// TIA Portal V17 export
// export: Created 2025-03-05T07:58:51.8164485Z, ExportSetting WithDefaults, DisplayName Totally Integrated Automation Portal, DisplayVersion V17 Update 8, DisplayName TIA Portal Openness, DisplayVersion V17 Update 8, DisplayName TIA Portal Version Control Interface, DisplayVersion V17, DisplayName SINAMICS Startdrive Advanced, DisplayVersion V17 SP2, DisplayName SINAMICS Startdrive G110M, G120, G120C, G120D, G120P, G115D, DisplayVersion V17 SP2, DisplayName SINAMICS Startdrive G130, G150, S120, S150, SINAMICS MV, S210, DisplayVersion V17 SP2, DisplayName STEP 7 Professional, DisplayVersion V17 Update 8, DisplayName SINUMERIK ONE STEP 7 Toolbox, DisplayVersion V17 Update 12, DisplayName SINUMERIK 840D sl STEP 7 Toolbox, DisplayVersion V17 Update 12, DisplayName STEP 7 Safety, DisplayVersion V17 Update 6, DisplayName WinCC Advanced, DisplayVersion V17 Update 8
DATA_BLOCK "LBP_CtrlEnergy"   // DB1000
TITLE = Ctrl-Energy
{ S7_Optimized_Access := 'FALSE'; DB_Accessible_From_OPC_UA := 'FALSE' }
AUTHOR : SINUMERIK
FAMILY : SINUMERIK_ONE
VERSION : 6.15
// Interface between user program and operating software, contains energy-saving profiles for Ctrl-Energy / La interfaz entre programa de usuario y software operativo, contiene perfiles de ahorro energético para Ctrl-Energy / Schnittstelle zwischen Anwenderprogramm und Betriebssoftware, enthält energiesparende Profile für Ctrl-Energy
// stored: AutoNumber false, DBAccessibleFromOPCUA false, DBAccessibleFromWebserver true, IsOnlyStoredInLoadMemory false, IsWriteProtectedInAS false
   VAR RETAIN
      Profile : Array[1..8] of Struct
         ESaveOn : Bool;   // Energiesparendes Profil sofort aktivieren / Activate energy-saving profile immediately / Activar inmediatamente perfil de ahorro energético
         ReloadT2 : Bool;   // Vorwarnzeit (T2) neu laden / Reload Prewarning time (T2) / Volver a cargar tiempo de prealarma (T2)
         res0_2 : Bool;
         res0_3 : Bool;
         res0_4 : Bool;
         res0_5 : Bool;
         res0_6 : Bool;
         res0_7 : Bool;
         HmiESaveOn : Bool;   // HMI->PLC: Energiesparendes Profil sofort aktivieren / HMI->PLC: Activate energy-saving profile immediately / HMI->PLC: activar inmediatamente perfil de ahorro energético
         res1_1 : Bool;
         res1_2 : Bool;
         res1_3 : Bool;
         res1_4 : Bool;
         res1_5 : Bool;
         res1_6 : Bool;
         res1_7 : Bool;
         MasterCompSig : Bool;   // Master-Rechner-Signal / Master computer signal / Señal de equipo maestro
         PlcUserSig : Bool;   // PLC-Anwendersignal / PLC user signal / Señal de usuario PLC
         res2_2 : Bool;
         res2_3 : Bool;
         res2_4 : Bool;
         res2_5 : Bool;
         res2_6 : Bool;
         res2_7 : Bool;
         res3 : Byte;
         ESaveIsOn : Bool;   // Energiesparender Zustand aktiv / Energy-saving state active / Estado de ahorro energético activo
         T1Expired : Bool;   // Aktivierungszeit T1 abgelaufen / Activation time T1 expired / Tiempo de activación T1 agotado
         res4_2 : Bool;
         res4_3 : Bool;
         res4_4 : Bool;
         res4_5 : Bool;
         res4_6 : Bool;
         res4_7 : Bool;
         res5 : Byte;
         ActValT1 : Int;   // T1 aktueller Wert / T1 current value / T1 valor actual
         ActValT2 : Int;   // T2 aktueller Wert / T2 current value / T2 valor actual
         ESaveValid : Bool;   // HMI->PLC: Energiesparendes Profil gültig / HMI->PLC: Energy-saving profile valid / HMI->PLC: perfil de ahorro energético válido
         ESaveOff : Bool;   // HMI->PLC: Energiesparendes Profil deaktivieren/sperren / HMI->PLC: Deactivate energy-saving profileblock energy-saving profile / HMI->PLC: activar/desactivar perfil de ahorro energético
         res10_2 : Bool;
         res10_3 : Bool;
         res10_4 : Bool;
         res10_5 : Bool;
         res10_6 : Bool;
         res10_7 : Bool;
         CondOpPanel : Bool;   // HMI->PLC: Bedienfeld / HMI->PLC: Operator panel / HMI->PLC: panel de mando
         CondDataTransfer : Bool;   // HMI->PLC: Datenübertragung / HMI->PLC: Data transfer / HMI->PLC: transferencia de datos
         CondWindowChange : Bool;   // HMI->PLC: Fensterwechsel / HMI->PLC: Window change / HMI->PLC: cambio de ventana
         res11_3 : Bool;
         res11_4 : Bool;
         res11_5 : Bool;
         res11_6 : Bool;
         res11_7 : Bool;
         CondMCP : Bool;   // HMI->PLC: Maschinen-Bedienfeld / HMI->PLC: Machine control panel / HMI->PLC: panel de mando de máquina
         res12_1 : Bool;
         res12_2 : Bool;
         res12_3 : Bool;
         res12_4 : Bool;
         res12_5 : Bool;
         res12_6 : Bool;
         res12_7 : Bool;
         CondNcChan1 : Bool;   // HMI->PLC: NC-Kanal 1 in Reset / HMI->PLC: NC channel 1 in reset / HMI->PLC: canal CN 1 en reset
         CondNcChan2 : Bool;   // HMI->PLC: NC-Kanal 2 in Reset / HMI->PLC: NC channel 2 in reset / HMI->PLC: canal CN 2 en reset
         CondNcChan3 : Bool;   // HMI->PLC: NC-Kanal 3 in Reset / HMI->PLC: NC channel 3 in reset / HMI->PLC: canal CN 3 en reset
         CondNcChan4 : Bool;   // HMI->PLC: NC-Kanal 4 in Reset / HMI->PLC: NC channel 4 in reset / HMI->PLC: canal CN 4 en reset
         CondNcChan5 : Bool;   // HMI->PLC: NC-Kanal 5 in Reset / HMI->PLC: NC channel 5 in reset / HMI->PLC: canal CN 5 en reset
         CondNcChan6 : Bool;   // HMI->PLC: NC-Kanal 6 in Reset / HMI->PLC: NC channel 6 in reset / HMI->PLC: canal CN 6 en reset
         CondNcChan7 : Bool;   // HMI->PLC: NC-Kanal 7 in Reset / HMI->PLC: NC channel 7 in reset / HMI->PLC: canal CN 7 en reset
         CondNcChan8 : Bool;   // HMI->PLC: NC-Kanal 8 in Reset / HMI->PLC: NC channel 8 in reset / HMI->PLC: canal CN 8 en reset
         CondNcChan9 : Bool;   // HMI->PLC: NC-Kanal 9 in Reset / HMI->PLC: NC channel 9 in reset / HMI->PLC: canal CN 9 en reset
         CondNcChan10 : Bool;   // HMI->PLC: NC-Kanal 10 in Reset / HMI->PLC: NC channel 10 in reset / HMI->PLC: canal CN 10 en reset
         res14_2 : Bool;
         res14_3 : Bool;
         res14_4 : Bool;
         res14_5 : Bool;
         res14_6 : Bool;
         res14_7 : Bool;
         CondMasterCompSig : Bool;   // HMI->PLC: Master-Rechner-Signal / HMI->PLC: Master computer signal / HMI->PLC: señal de equipo maestro
         CondPlcUserSig : Bool;   // HMI->PLC: PLC-Anwendersignal / HMI->PLC: PLC user signal / HMI->PLC: señal de usuario PLC
         res15_2 : Bool;
         res15_3 : Bool;
         res15_4 : Bool;
         res15_5 : Bool;
         res15_6 : Bool;
         res15_7 : Bool;
         PresetT1 : Int;   // HMI->PLC: Aktivierung Zeit T1 / HMI->PLC: Activation time T1 / HMI->PLC: activación tiempo T1
         PresetT2 : Int;   // HMI->PLC: Vorwarnzeit T2 / HMI->PLC: Prewarning time T2 / HMI->PLC: tiempo de prealarma T2
      END_STRUCT;
   END_VAR
BEGIN
   // Profile[2].ESaveOn : Energiesparendes Profil sofort aktivieren / Activate energy-saving profile immediately / Activar inmediatamente perfil de ahorro energético
   // Profile[3].ESaveOn : Energiesparendes Profil sofort aktivieren / Activate energy-saving profile immediately / Activar inmediatamente perfil de ahorro energético
   // Profile[4].ESaveOn : Energiesparendes Profil sofort aktivieren / Activate energy-saving profile immediately / Activar inmediatamente perfil de ahorro energético
   // Profile[5].ESaveOn : Energiesparendes Profil sofort aktivieren / Activate energy-saving profile immediately / Activar inmediatamente perfil de ahorro energético
   // Profile[6].ESaveOn : Energiesparendes Profil sofort aktivieren / Activate energy-saving profile immediately / Activar inmediatamente perfil de ahorro energético
   // Profile[7].ESaveOn : Energiesparendes Profil sofort aktivieren / Activate energy-saving profile immediately / Activar inmediatamente perfil de ahorro energético
   // Profile[8].ESaveOn : Energiesparendes Profil sofort aktivieren / Activate energy-saving profile immediately / Activar inmediatamente perfil de ahorro energético
   // Profile[2].ReloadT2 : Vorwarnzeit (T2) neu laden / Reload Prewarning time (T2) / Volver a cargar tiempo de prealarma (T2)
   // Profile[3].ReloadT2 : Vorwarnzeit (T2) neu laden / Reload Prewarning time (T2) / Volver a cargar tiempo de prealarma (T2)
   // Profile[4].ReloadT2 : Vorwarnzeit (T2) neu laden / Reload Prewarning time (T2) / Volver a cargar tiempo de prealarma (T2)
   // Profile[5].ReloadT2 : Vorwarnzeit (T2) neu laden / Reload Prewarning time (T2) / Volver a cargar tiempo de prealarma (T2)
   // Profile[6].ReloadT2 : Vorwarnzeit (T2) neu laden / Reload Prewarning time (T2) / Volver a cargar tiempo de prealarma (T2)
   // Profile[7].ReloadT2 : Vorwarnzeit (T2) neu laden / Reload Prewarning time (T2) / Volver a cargar tiempo de prealarma (T2)
   // Profile[8].ReloadT2 : Vorwarnzeit (T2) neu laden / Reload Prewarning time (T2) / Volver a cargar tiempo de prealarma (T2)
   // Profile[2].HmiESaveOn : HMI->PLC: Energiesparendes Profil sofort aktivieren / HMI->PLC: Activate energy-saving profile immediately / HMI->PLC: activar inmediatamente perfil de ahorro energético
   // Profile[3].HmiESaveOn : HMI->PLC: Energiesparendes Profil sofort aktivieren / HMI->PLC: Activate energy-saving profile immediately / HMI->PLC: activar inmediatamente perfil de ahorro energético
   // Profile[4].HmiESaveOn : HMI->PLC: Energiesparendes Profil sofort aktivieren / HMI->PLC: Activate energy-saving profile immediately / HMI->PLC: activar inmediatamente perfil de ahorro energético
   // Profile[5].HmiESaveOn : HMI->PLC: Energiesparendes Profil sofort aktivieren / HMI->PLC: Activate energy-saving profile immediately / HMI->PLC: activar inmediatamente perfil de ahorro energético
   // Profile[6].HmiESaveOn : HMI->PLC: Energiesparendes Profil sofort aktivieren / HMI->PLC: Activate energy-saving profile immediately / HMI->PLC: activar inmediatamente perfil de ahorro energético
   // Profile[7].HmiESaveOn : HMI->PLC: Energiesparendes Profil sofort aktivieren / HMI->PLC: Activate energy-saving profile immediately / HMI->PLC: activar inmediatamente perfil de ahorro energético
   // Profile[8].HmiESaveOn : HMI->PLC: Energiesparendes Profil sofort aktivieren / HMI->PLC: Activate energy-saving profile immediately / HMI->PLC: activar inmediatamente perfil de ahorro energético
   // Profile[2].MasterCompSig : Master-Rechner-Signal / Master computer signal / Señal de equipo maestro
   // Profile[3].MasterCompSig : Master-Rechner-Signal / Master computer signal / Señal de equipo maestro
   // Profile[4].MasterCompSig : Master-Rechner-Signal / Master computer signal / Señal de equipo maestro
   // Profile[5].MasterCompSig : Master-Rechner-Signal / Master computer signal / Señal de equipo maestro
   // Profile[6].MasterCompSig : Master-Rechner-Signal / Master computer signal / Señal de equipo maestro
   // Profile[7].MasterCompSig : Master-Rechner-Signal / Master computer signal / Señal de equipo maestro
   // Profile[8].MasterCompSig : Master-Rechner-Signal / Master computer signal / Señal de equipo maestro
   // Profile[2].PlcUserSig : PLC-Anwendersignal / PLC user signal / Señal de usuario PLC
   // Profile[3].PlcUserSig : PLC-Anwendersignal / PLC user signal / Señal de usuario PLC
   // Profile[4].PlcUserSig : PLC-Anwendersignal / PLC user signal / Señal de usuario PLC
   // Profile[5].PlcUserSig : PLC-Anwendersignal / PLC user signal / Señal de usuario PLC
   // Profile[6].PlcUserSig : PLC-Anwendersignal / PLC user signal / Señal de usuario PLC
   // Profile[7].PlcUserSig : PLC-Anwendersignal / PLC user signal / Señal de usuario PLC
   // Profile[8].PlcUserSig : PLC-Anwendersignal / PLC user signal / Señal de usuario PLC
   // Profile[2].ESaveIsOn : Energiesparender Zustand aktiv / Energy-saving state active / Estado de ahorro energético activo
   // Profile[3].ESaveIsOn : Energiesparender Zustand aktiv / Energy-saving state active / Estado de ahorro energético activo
   // Profile[4].ESaveIsOn : Energiesparender Zustand aktiv / Energy-saving state active / Estado de ahorro energético activo
   // Profile[5].ESaveIsOn : Energiesparender Zustand aktiv / Energy-saving state active / Estado de ahorro energético activo
   // Profile[6].ESaveIsOn : Energiesparender Zustand aktiv / Energy-saving state active / Estado de ahorro energético activo
   // Profile[7].ESaveIsOn : Energiesparender Zustand aktiv / Energy-saving state active / Estado de ahorro energético activo
   // Profile[8].ESaveIsOn : Energiesparender Zustand aktiv / Energy-saving state active / Estado de ahorro energético activo
   // Profile[2].T1Expired : Aktivierungszeit T1 abgelaufen / Activation time T1 expired / Tiempo de activación T1 agotado
   // Profile[3].T1Expired : Aktivierungszeit T1 abgelaufen / Activation time T1 expired / Tiempo de activación T1 agotado
   // Profile[4].T1Expired : Aktivierungszeit T1 abgelaufen / Activation time T1 expired / Tiempo de activación T1 agotado
   // Profile[5].T1Expired : Aktivierungszeit T1 abgelaufen / Activation time T1 expired / Tiempo de activación T1 agotado
   // Profile[6].T1Expired : Aktivierungszeit T1 abgelaufen / Activation time T1 expired / Tiempo de activación T1 agotado
   // Profile[7].T1Expired : Aktivierungszeit T1 abgelaufen / Activation time T1 expired / Tiempo de activación T1 agotado
   // Profile[8].T1Expired : Aktivierungszeit T1 abgelaufen / Activation time T1 expired / Tiempo de activación T1 agotado
   // Profile[2].ActValT1 : T1 aktueller Wert / T1 current value / T1 valor actual
   // Profile[3].ActValT1 : T1 aktueller Wert / T1 current value / T1 valor actual
   // Profile[4].ActValT1 : T1 aktueller Wert / T1 current value / T1 valor actual
   // Profile[5].ActValT1 : T1 aktueller Wert / T1 current value / T1 valor actual
   // Profile[6].ActValT1 : T1 aktueller Wert / T1 current value / T1 valor actual
   // Profile[7].ActValT1 : T1 aktueller Wert / T1 current value / T1 valor actual
   // Profile[8].ActValT1 : T1 aktueller Wert / T1 current value / T1 valor actual
   // Profile[2].ActValT2 : T2 aktueller Wert / T2 current value / T2 valor actual
   // Profile[3].ActValT2 : T2 aktueller Wert / T2 current value / T2 valor actual
   // Profile[4].ActValT2 : T2 aktueller Wert / T2 current value / T2 valor actual
   // Profile[5].ActValT2 : T2 aktueller Wert / T2 current value / T2 valor actual
   // Profile[6].ActValT2 : T2 aktueller Wert / T2 current value / T2 valor actual
   // Profile[7].ActValT2 : T2 aktueller Wert / T2 current value / T2 valor actual
   // Profile[8].ActValT2 : T2 aktueller Wert / T2 current value / T2 valor actual
   Profile[1].ESaveValid := TRUE;
   Profile[2].ESaveValid := TRUE;   // HMI->PLC: Energiesparendes Profil gültig / HMI->PLC: Energy-saving profile valid / HMI->PLC: perfil de ahorro energético válido
   Profile[3].ESaveValid := TRUE;   // HMI->PLC: Energiesparendes Profil gültig / HMI->PLC: Energy-saving profile valid / HMI->PLC: perfil de ahorro energético válido
   // Profile[4].ESaveValid : HMI->PLC: Energiesparendes Profil gültig / HMI->PLC: Energy-saving profile valid / HMI->PLC: perfil de ahorro energético válido
   // Profile[5].ESaveValid : HMI->PLC: Energiesparendes Profil gültig / HMI->PLC: Energy-saving profile valid / HMI->PLC: perfil de ahorro energético válido
   // Profile[6].ESaveValid : HMI->PLC: Energiesparendes Profil gültig / HMI->PLC: Energy-saving profile valid / HMI->PLC: perfil de ahorro energético válido
   // Profile[7].ESaveValid : HMI->PLC: Energiesparendes Profil gültig / HMI->PLC: Energy-saving profile valid / HMI->PLC: perfil de ahorro energético válido
   // Profile[8].ESaveValid : HMI->PLC: Energiesparendes Profil gültig / HMI->PLC: Energy-saving profile valid / HMI->PLC: perfil de ahorro energético válido
   Profile[1].ESaveOff := TRUE;
   Profile[2].ESaveOff := TRUE;   // HMI->PLC: Energiesparendes Profil deaktivieren/sperren / HMI->PLC: Deactivate energy-saving profileblock energy-saving profile / HMI->PLC: activar/desactivar perfil de ahorro energético
   Profile[3].ESaveOff := TRUE;   // HMI->PLC: Energiesparendes Profil deaktivieren/sperren / HMI->PLC: Deactivate energy-saving profileblock energy-saving profile / HMI->PLC: activar/desactivar perfil de ahorro energético
   // Profile[4].ESaveOff : HMI->PLC: Energiesparendes Profil deaktivieren/sperren / HMI->PLC: Deactivate energy-saving profileblock energy-saving profile / HMI->PLC: activar/desactivar perfil de ahorro energético
   // Profile[5].ESaveOff : HMI->PLC: Energiesparendes Profil deaktivieren/sperren / HMI->PLC: Deactivate energy-saving profileblock energy-saving profile / HMI->PLC: activar/desactivar perfil de ahorro energético
   // Profile[6].ESaveOff : HMI->PLC: Energiesparendes Profil deaktivieren/sperren / HMI->PLC: Deactivate energy-saving profileblock energy-saving profile / HMI->PLC: activar/desactivar perfil de ahorro energético
   // Profile[7].ESaveOff : HMI->PLC: Energiesparendes Profil deaktivieren/sperren / HMI->PLC: Deactivate energy-saving profileblock energy-saving profile / HMI->PLC: activar/desactivar perfil de ahorro energético
   // Profile[8].ESaveOff : HMI->PLC: Energiesparendes Profil deaktivieren/sperren / HMI->PLC: Deactivate energy-saving profileblock energy-saving profile / HMI->PLC: activar/desactivar perfil de ahorro energético
   // Profile[2].CondOpPanel : HMI->PLC: Bedienfeld / HMI->PLC: Operator panel / HMI->PLC: panel de mando
   Profile[3].CondOpPanel := TRUE;   // HMI->PLC: Bedienfeld / HMI->PLC: Operator panel / HMI->PLC: panel de mando
   // Profile[4].CondOpPanel : HMI->PLC: Bedienfeld / HMI->PLC: Operator panel / HMI->PLC: panel de mando
   // Profile[5].CondOpPanel : HMI->PLC: Bedienfeld / HMI->PLC: Operator panel / HMI->PLC: panel de mando
   // Profile[6].CondOpPanel : HMI->PLC: Bedienfeld / HMI->PLC: Operator panel / HMI->PLC: panel de mando
   // Profile[7].CondOpPanel : HMI->PLC: Bedienfeld / HMI->PLC: Operator panel / HMI->PLC: panel de mando
   // Profile[8].CondOpPanel : HMI->PLC: Bedienfeld / HMI->PLC: Operator panel / HMI->PLC: panel de mando
   // Profile[2].CondDataTransfer : HMI->PLC: Datenübertragung / HMI->PLC: Data transfer / HMI->PLC: transferencia de datos
   Profile[3].CondDataTransfer := TRUE;   // HMI->PLC: Datenübertragung / HMI->PLC: Data transfer / HMI->PLC: transferencia de datos
   // Profile[4].CondDataTransfer : HMI->PLC: Datenübertragung / HMI->PLC: Data transfer / HMI->PLC: transferencia de datos
   // Profile[5].CondDataTransfer : HMI->PLC: Datenübertragung / HMI->PLC: Data transfer / HMI->PLC: transferencia de datos
   // Profile[6].CondDataTransfer : HMI->PLC: Datenübertragung / HMI->PLC: Data transfer / HMI->PLC: transferencia de datos
   // Profile[7].CondDataTransfer : HMI->PLC: Datenübertragung / HMI->PLC: Data transfer / HMI->PLC: transferencia de datos
   // Profile[8].CondDataTransfer : HMI->PLC: Datenübertragung / HMI->PLC: Data transfer / HMI->PLC: transferencia de datos
   // Profile[2].CondWindowChange : HMI->PLC: Fensterwechsel / HMI->PLC: Window change / HMI->PLC: cambio de ventana
   Profile[3].CondWindowChange := TRUE;   // HMI->PLC: Fensterwechsel / HMI->PLC: Window change / HMI->PLC: cambio de ventana
   // Profile[4].CondWindowChange : HMI->PLC: Fensterwechsel / HMI->PLC: Window change / HMI->PLC: cambio de ventana
   // Profile[5].CondWindowChange : HMI->PLC: Fensterwechsel / HMI->PLC: Window change / HMI->PLC: cambio de ventana
   // Profile[6].CondWindowChange : HMI->PLC: Fensterwechsel / HMI->PLC: Window change / HMI->PLC: cambio de ventana
   // Profile[7].CondWindowChange : HMI->PLC: Fensterwechsel / HMI->PLC: Window change / HMI->PLC: cambio de ventana
   // Profile[8].CondWindowChange : HMI->PLC: Fensterwechsel / HMI->PLC: Window change / HMI->PLC: cambio de ventana
   Profile[2].CondMCP := TRUE;   // HMI->PLC: Maschinen-Bedienfeld / HMI->PLC: Machine control panel / HMI->PLC: panel de mando de máquina
   Profile[3].CondMCP := TRUE;   // HMI->PLC: Maschinen-Bedienfeld / HMI->PLC: Machine control panel / HMI->PLC: panel de mando de máquina
   // Profile[4].CondMCP : HMI->PLC: Maschinen-Bedienfeld / HMI->PLC: Machine control panel / HMI->PLC: panel de mando de máquina
   // Profile[5].CondMCP : HMI->PLC: Maschinen-Bedienfeld / HMI->PLC: Machine control panel / HMI->PLC: panel de mando de máquina
   // Profile[6].CondMCP : HMI->PLC: Maschinen-Bedienfeld / HMI->PLC: Machine control panel / HMI->PLC: panel de mando de máquina
   // Profile[7].CondMCP : HMI->PLC: Maschinen-Bedienfeld / HMI->PLC: Machine control panel / HMI->PLC: panel de mando de máquina
   // Profile[8].CondMCP : HMI->PLC: Maschinen-Bedienfeld / HMI->PLC: Machine control panel / HMI->PLC: panel de mando de máquina
   Profile[1].CondNcChan1 := TRUE;
   Profile[2].CondNcChan1 := TRUE;   // HMI->PLC: NC-Kanal 1 in Reset / HMI->PLC: NC channel 1 in reset / HMI->PLC: canal CN 1 en reset
   Profile[3].CondNcChan1 := TRUE;   // HMI->PLC: NC-Kanal 1 in Reset / HMI->PLC: NC channel 1 in reset / HMI->PLC: canal CN 1 en reset
   // Profile[4].CondNcChan1 : HMI->PLC: NC-Kanal 1 in Reset / HMI->PLC: NC channel 1 in reset / HMI->PLC: canal CN 1 en reset
   // Profile[5].CondNcChan1 : HMI->PLC: NC-Kanal 1 in Reset / HMI->PLC: NC channel 1 in reset / HMI->PLC: canal CN 1 en reset
   // Profile[6].CondNcChan1 : HMI->PLC: NC-Kanal 1 in Reset / HMI->PLC: NC channel 1 in reset / HMI->PLC: canal CN 1 en reset
   // Profile[7].CondNcChan1 : HMI->PLC: NC-Kanal 1 in Reset / HMI->PLC: NC channel 1 in reset / HMI->PLC: canal CN 1 en reset
   // Profile[8].CondNcChan1 : HMI->PLC: NC-Kanal 1 in Reset / HMI->PLC: NC channel 1 in reset / HMI->PLC: canal CN 1 en reset
   Profile[1].CondNcChan2 := TRUE;
   Profile[2].CondNcChan2 := TRUE;   // HMI->PLC: NC-Kanal 2 in Reset / HMI->PLC: NC channel 2 in reset / HMI->PLC: canal CN 2 en reset
   Profile[3].CondNcChan2 := TRUE;   // HMI->PLC: NC-Kanal 2 in Reset / HMI->PLC: NC channel 2 in reset / HMI->PLC: canal CN 2 en reset
   // Profile[4].CondNcChan2 : HMI->PLC: NC-Kanal 2 in Reset / HMI->PLC: NC channel 2 in reset / HMI->PLC: canal CN 2 en reset
   // Profile[5].CondNcChan2 : HMI->PLC: NC-Kanal 2 in Reset / HMI->PLC: NC channel 2 in reset / HMI->PLC: canal CN 2 en reset
   // Profile[6].CondNcChan2 : HMI->PLC: NC-Kanal 2 in Reset / HMI->PLC: NC channel 2 in reset / HMI->PLC: canal CN 2 en reset
   // Profile[7].CondNcChan2 : HMI->PLC: NC-Kanal 2 in Reset / HMI->PLC: NC channel 2 in reset / HMI->PLC: canal CN 2 en reset
   // Profile[8].CondNcChan2 : HMI->PLC: NC-Kanal 2 in Reset / HMI->PLC: NC channel 2 in reset / HMI->PLC: canal CN 2 en reset
   Profile[1].CondNcChan3 := TRUE;
   Profile[2].CondNcChan3 := TRUE;   // HMI->PLC: NC-Kanal 3 in Reset / HMI->PLC: NC channel 3 in reset / HMI->PLC: canal CN 3 en reset
   Profile[3].CondNcChan3 := TRUE;   // HMI->PLC: NC-Kanal 3 in Reset / HMI->PLC: NC channel 3 in reset / HMI->PLC: canal CN 3 en reset
   // Profile[4].CondNcChan3 : HMI->PLC: NC-Kanal 3 in Reset / HMI->PLC: NC channel 3 in reset / HMI->PLC: canal CN 3 en reset
   // Profile[5].CondNcChan3 : HMI->PLC: NC-Kanal 3 in Reset / HMI->PLC: NC channel 3 in reset / HMI->PLC: canal CN 3 en reset
   // Profile[6].CondNcChan3 : HMI->PLC: NC-Kanal 3 in Reset / HMI->PLC: NC channel 3 in reset / HMI->PLC: canal CN 3 en reset
   // Profile[7].CondNcChan3 : HMI->PLC: NC-Kanal 3 in Reset / HMI->PLC: NC channel 3 in reset / HMI->PLC: canal CN 3 en reset
   // Profile[8].CondNcChan3 : HMI->PLC: NC-Kanal 3 in Reset / HMI->PLC: NC channel 3 in reset / HMI->PLC: canal CN 3 en reset
   Profile[1].CondNcChan4 := TRUE;
   Profile[2].CondNcChan4 := TRUE;   // HMI->PLC: NC-Kanal 4 in Reset / HMI->PLC: NC channel 4 in reset / HMI->PLC: canal CN 4 en reset
   Profile[3].CondNcChan4 := TRUE;   // HMI->PLC: NC-Kanal 4 in Reset / HMI->PLC: NC channel 4 in reset / HMI->PLC: canal CN 4 en reset
   // Profile[4].CondNcChan4 : HMI->PLC: NC-Kanal 4 in Reset / HMI->PLC: NC channel 4 in reset / HMI->PLC: canal CN 4 en reset
   // Profile[5].CondNcChan4 : HMI->PLC: NC-Kanal 4 in Reset / HMI->PLC: NC channel 4 in reset / HMI->PLC: canal CN 4 en reset
   // Profile[6].CondNcChan4 : HMI->PLC: NC-Kanal 4 in Reset / HMI->PLC: NC channel 4 in reset / HMI->PLC: canal CN 4 en reset
   // Profile[7].CondNcChan4 : HMI->PLC: NC-Kanal 4 in Reset / HMI->PLC: NC channel 4 in reset / HMI->PLC: canal CN 4 en reset
   // Profile[8].CondNcChan4 : HMI->PLC: NC-Kanal 4 in Reset / HMI->PLC: NC channel 4 in reset / HMI->PLC: canal CN 4 en reset
   Profile[1].CondNcChan5 := TRUE;
   Profile[2].CondNcChan5 := TRUE;   // HMI->PLC: NC-Kanal 5 in Reset / HMI->PLC: NC channel 5 in reset / HMI->PLC: canal CN 5 en reset
   Profile[3].CondNcChan5 := TRUE;   // HMI->PLC: NC-Kanal 5 in Reset / HMI->PLC: NC channel 5 in reset / HMI->PLC: canal CN 5 en reset
   // Profile[4].CondNcChan5 : HMI->PLC: NC-Kanal 5 in Reset / HMI->PLC: NC channel 5 in reset / HMI->PLC: canal CN 5 en reset
   // Profile[5].CondNcChan5 : HMI->PLC: NC-Kanal 5 in Reset / HMI->PLC: NC channel 5 in reset / HMI->PLC: canal CN 5 en reset
   // Profile[6].CondNcChan5 : HMI->PLC: NC-Kanal 5 in Reset / HMI->PLC: NC channel 5 in reset / HMI->PLC: canal CN 5 en reset
   // Profile[7].CondNcChan5 : HMI->PLC: NC-Kanal 5 in Reset / HMI->PLC: NC channel 5 in reset / HMI->PLC: canal CN 5 en reset
   // Profile[8].CondNcChan5 : HMI->PLC: NC-Kanal 5 in Reset / HMI->PLC: NC channel 5 in reset / HMI->PLC: canal CN 5 en reset
   Profile[1].CondNcChan6 := TRUE;
   Profile[2].CondNcChan6 := TRUE;   // HMI->PLC: NC-Kanal 6 in Reset / HMI->PLC: NC channel 6 in reset / HMI->PLC: canal CN 6 en reset
   Profile[3].CondNcChan6 := TRUE;   // HMI->PLC: NC-Kanal 6 in Reset / HMI->PLC: NC channel 6 in reset / HMI->PLC: canal CN 6 en reset
   // Profile[4].CondNcChan6 : HMI->PLC: NC-Kanal 6 in Reset / HMI->PLC: NC channel 6 in reset / HMI->PLC: canal CN 6 en reset
   // Profile[5].CondNcChan6 : HMI->PLC: NC-Kanal 6 in Reset / HMI->PLC: NC channel 6 in reset / HMI->PLC: canal CN 6 en reset
   // Profile[6].CondNcChan6 : HMI->PLC: NC-Kanal 6 in Reset / HMI->PLC: NC channel 6 in reset / HMI->PLC: canal CN 6 en reset
   // Profile[7].CondNcChan6 : HMI->PLC: NC-Kanal 6 in Reset / HMI->PLC: NC channel 6 in reset / HMI->PLC: canal CN 6 en reset
   // Profile[8].CondNcChan6 : HMI->PLC: NC-Kanal 6 in Reset / HMI->PLC: NC channel 6 in reset / HMI->PLC: canal CN 6 en reset
   Profile[1].CondNcChan7 := TRUE;
   Profile[2].CondNcChan7 := TRUE;   // HMI->PLC: NC-Kanal 7 in Reset / HMI->PLC: NC channel 7 in reset / HMI->PLC: canal CN 7 en reset
   Profile[3].CondNcChan7 := TRUE;   // HMI->PLC: NC-Kanal 7 in Reset / HMI->PLC: NC channel 7 in reset / HMI->PLC: canal CN 7 en reset
   // Profile[4].CondNcChan7 : HMI->PLC: NC-Kanal 7 in Reset / HMI->PLC: NC channel 7 in reset / HMI->PLC: canal CN 7 en reset
   // Profile[5].CondNcChan7 : HMI->PLC: NC-Kanal 7 in Reset / HMI->PLC: NC channel 7 in reset / HMI->PLC: canal CN 7 en reset
   // Profile[6].CondNcChan7 : HMI->PLC: NC-Kanal 7 in Reset / HMI->PLC: NC channel 7 in reset / HMI->PLC: canal CN 7 en reset
   // Profile[7].CondNcChan7 : HMI->PLC: NC-Kanal 7 in Reset / HMI->PLC: NC channel 7 in reset / HMI->PLC: canal CN 7 en reset
   // Profile[8].CondNcChan7 : HMI->PLC: NC-Kanal 7 in Reset / HMI->PLC: NC channel 7 in reset / HMI->PLC: canal CN 7 en reset
   Profile[1].CondNcChan8 := TRUE;
   Profile[2].CondNcChan8 := TRUE;   // HMI->PLC: NC-Kanal 8 in Reset / HMI->PLC: NC channel 8 in reset / HMI->PLC: canal CN 8 en reset
   Profile[3].CondNcChan8 := TRUE;   // HMI->PLC: NC-Kanal 8 in Reset / HMI->PLC: NC channel 8 in reset / HMI->PLC: canal CN 8 en reset
   // Profile[4].CondNcChan8 : HMI->PLC: NC-Kanal 8 in Reset / HMI->PLC: NC channel 8 in reset / HMI->PLC: canal CN 8 en reset
   // Profile[5].CondNcChan8 : HMI->PLC: NC-Kanal 8 in Reset / HMI->PLC: NC channel 8 in reset / HMI->PLC: canal CN 8 en reset
   // Profile[6].CondNcChan8 : HMI->PLC: NC-Kanal 8 in Reset / HMI->PLC: NC channel 8 in reset / HMI->PLC: canal CN 8 en reset
   // Profile[7].CondNcChan8 : HMI->PLC: NC-Kanal 8 in Reset / HMI->PLC: NC channel 8 in reset / HMI->PLC: canal CN 8 en reset
   // Profile[8].CondNcChan8 : HMI->PLC: NC-Kanal 8 in Reset / HMI->PLC: NC channel 8 in reset / HMI->PLC: canal CN 8 en reset
   Profile[1].CondNcChan9 := TRUE;
   Profile[2].CondNcChan9 := TRUE;   // HMI->PLC: NC-Kanal 9 in Reset / HMI->PLC: NC channel 9 in reset / HMI->PLC: canal CN 9 en reset
   Profile[3].CondNcChan9 := TRUE;   // HMI->PLC: NC-Kanal 9 in Reset / HMI->PLC: NC channel 9 in reset / HMI->PLC: canal CN 9 en reset
   // Profile[4].CondNcChan9 : HMI->PLC: NC-Kanal 9 in Reset / HMI->PLC: NC channel 9 in reset / HMI->PLC: canal CN 9 en reset
   // Profile[5].CondNcChan9 : HMI->PLC: NC-Kanal 9 in Reset / HMI->PLC: NC channel 9 in reset / HMI->PLC: canal CN 9 en reset
   // Profile[6].CondNcChan9 : HMI->PLC: NC-Kanal 9 in Reset / HMI->PLC: NC channel 9 in reset / HMI->PLC: canal CN 9 en reset
   // Profile[7].CondNcChan9 : HMI->PLC: NC-Kanal 9 in Reset / HMI->PLC: NC channel 9 in reset / HMI->PLC: canal CN 9 en reset
   // Profile[8].CondNcChan9 : HMI->PLC: NC-Kanal 9 in Reset / HMI->PLC: NC channel 9 in reset / HMI->PLC: canal CN 9 en reset
   Profile[1].CondNcChan10 := TRUE;
   Profile[2].CondNcChan10 := TRUE;   // HMI->PLC: NC-Kanal 10 in Reset / HMI->PLC: NC channel 10 in reset / HMI->PLC: canal CN 10 en reset
   Profile[3].CondNcChan10 := TRUE;   // HMI->PLC: NC-Kanal 10 in Reset / HMI->PLC: NC channel 10 in reset / HMI->PLC: canal CN 10 en reset
   // Profile[4].CondNcChan10 : HMI->PLC: NC-Kanal 10 in Reset / HMI->PLC: NC channel 10 in reset / HMI->PLC: canal CN 10 en reset
   // Profile[5].CondNcChan10 : HMI->PLC: NC-Kanal 10 in Reset / HMI->PLC: NC channel 10 in reset / HMI->PLC: canal CN 10 en reset
   // Profile[6].CondNcChan10 : HMI->PLC: NC-Kanal 10 in Reset / HMI->PLC: NC channel 10 in reset / HMI->PLC: canal CN 10 en reset
   // Profile[7].CondNcChan10 : HMI->PLC: NC-Kanal 10 in Reset / HMI->PLC: NC channel 10 in reset / HMI->PLC: canal CN 10 en reset
   // Profile[8].CondNcChan10 : HMI->PLC: NC-Kanal 10 in Reset / HMI->PLC: NC channel 10 in reset / HMI->PLC: canal CN 10 en reset
   // Profile[2].CondMasterCompSig : HMI->PLC: Master-Rechner-Signal / HMI->PLC: Master computer signal / HMI->PLC: señal de equipo maestro
   // Profile[3].CondMasterCompSig : HMI->PLC: Master-Rechner-Signal / HMI->PLC: Master computer signal / HMI->PLC: señal de equipo maestro
   // Profile[4].CondMasterCompSig : HMI->PLC: Master-Rechner-Signal / HMI->PLC: Master computer signal / HMI->PLC: señal de equipo maestro
   // Profile[5].CondMasterCompSig : HMI->PLC: Master-Rechner-Signal / HMI->PLC: Master computer signal / HMI->PLC: señal de equipo maestro
   // Profile[6].CondMasterCompSig : HMI->PLC: Master-Rechner-Signal / HMI->PLC: Master computer signal / HMI->PLC: señal de equipo maestro
   // Profile[7].CondMasterCompSig : HMI->PLC: Master-Rechner-Signal / HMI->PLC: Master computer signal / HMI->PLC: señal de equipo maestro
   // Profile[8].CondMasterCompSig : HMI->PLC: Master-Rechner-Signal / HMI->PLC: Master computer signal / HMI->PLC: señal de equipo maestro
   Profile[1].CondPlcUserSig := TRUE;
   Profile[2].CondPlcUserSig := TRUE;   // HMI->PLC: PLC-Anwendersignal / HMI->PLC: PLC user signal / HMI->PLC: señal de usuario PLC
   Profile[3].CondPlcUserSig := TRUE;   // HMI->PLC: PLC-Anwendersignal / HMI->PLC: PLC user signal / HMI->PLC: señal de usuario PLC
   // Profile[4].CondPlcUserSig : HMI->PLC: PLC-Anwendersignal / HMI->PLC: PLC user signal / HMI->PLC: señal de usuario PLC
   // Profile[5].CondPlcUserSig : HMI->PLC: PLC-Anwendersignal / HMI->PLC: PLC user signal / HMI->PLC: señal de usuario PLC
   // Profile[6].CondPlcUserSig : HMI->PLC: PLC-Anwendersignal / HMI->PLC: PLC user signal / HMI->PLC: señal de usuario PLC
   // Profile[7].CondPlcUserSig : HMI->PLC: PLC-Anwendersignal / HMI->PLC: PLC user signal / HMI->PLC: señal de usuario PLC
   // Profile[8].CondPlcUserSig : HMI->PLC: PLC-Anwendersignal / HMI->PLC: PLC user signal / HMI->PLC: señal de usuario PLC
   Profile[1].PresetT1 := 60;
   Profile[2].PresetT1 := 120;   // HMI->PLC: Aktivierung Zeit T1 / HMI->PLC: Activation time T1 / HMI->PLC: activación tiempo T1
   Profile[3].PresetT1 := 600;   // HMI->PLC: Aktivierung Zeit T1 / HMI->PLC: Activation time T1 / HMI->PLC: activación tiempo T1
   // Profile[4].PresetT1 : HMI->PLC: Aktivierung Zeit T1 / HMI->PLC: Activation time T1 / HMI->PLC: activación tiempo T1
   // Profile[5].PresetT1 : HMI->PLC: Aktivierung Zeit T1 / HMI->PLC: Activation time T1 / HMI->PLC: activación tiempo T1
   // Profile[6].PresetT1 : HMI->PLC: Aktivierung Zeit T1 / HMI->PLC: Activation time T1 / HMI->PLC: activación tiempo T1
   // Profile[7].PresetT1 : HMI->PLC: Aktivierung Zeit T1 / HMI->PLC: Activation time T1 / HMI->PLC: activación tiempo T1
   // Profile[8].PresetT1 : HMI->PLC: Aktivierung Zeit T1 / HMI->PLC: Activation time T1 / HMI->PLC: activación tiempo T1
   Profile[1].PresetT2 := 120;
   Profile[2].PresetT2 := 300;   // HMI->PLC: Vorwarnzeit T2 / HMI->PLC: Prewarning time T2 / HMI->PLC: tiempo de prealarma T2
   // Profile[3].PresetT2 : HMI->PLC: Vorwarnzeit T2 / HMI->PLC: Prewarning time T2 / HMI->PLC: tiempo de prealarma T2
   // Profile[4].PresetT2 : HMI->PLC: Vorwarnzeit T2 / HMI->PLC: Prewarning time T2 / HMI->PLC: tiempo de prealarma T2
   // Profile[5].PresetT2 : HMI->PLC: Vorwarnzeit T2 / HMI->PLC: Prewarning time T2 / HMI->PLC: tiempo de prealarma T2
   // Profile[6].PresetT2 : HMI->PLC: Vorwarnzeit T2 / HMI->PLC: Prewarning time T2 / HMI->PLC: tiempo de prealarma T2
   // Profile[7].PresetT2 : HMI->PLC: Vorwarnzeit T2 / HMI->PLC: Prewarning time T2 / HMI->PLC: tiempo de prealarma T2
   // Profile[8].PresetT2 : HMI->PLC: Vorwarnzeit T2 / HMI->PLC: Prewarning time T2 / HMI->PLC: tiempo de prealarma T2
END_DATA_BLOCK
